RoboDK station: NiryoStation.rdk

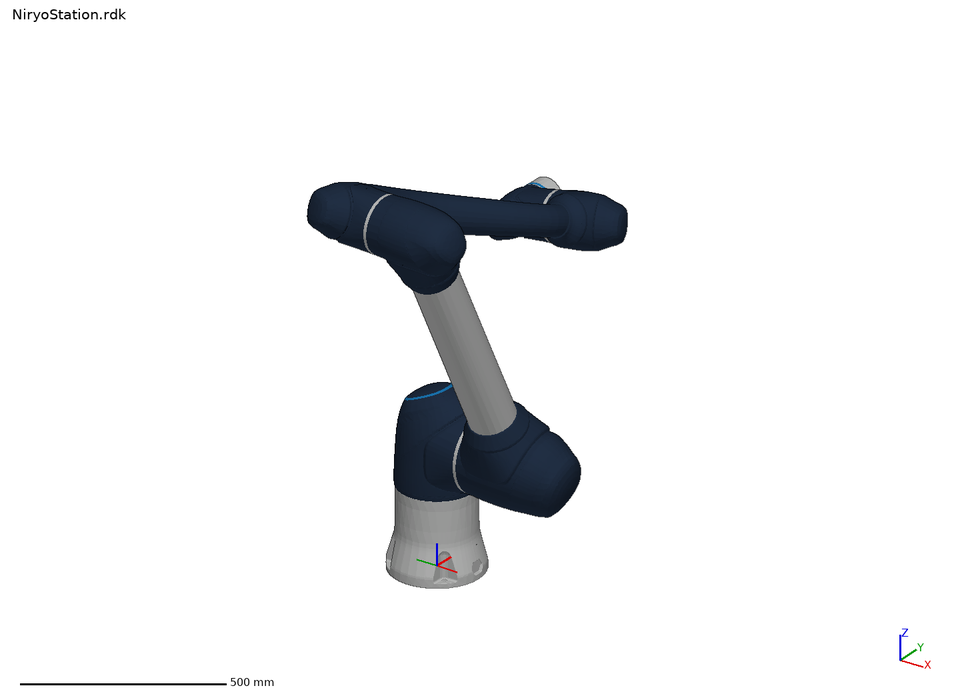
[picture v0: the station drawn from its stored meshes, robots at their saved joint values, targets as dots, program paths as lines]
Station NiryoStation (saved by RoboDK 5.5.1). Poses are relative to the parent item; angles as X-Y-Z fixed-axis rotations.
  - frame wall at (0, 0, 0) mm
    - frame RoboBase at (0, 0, 0) mm, rotated rx 0 ry 0 rz 90 deg
      - robot Doosan Robotics H2017: 6 axes, payload 20 kg, reach 1700 mm, repeatability 0.1 mm
          modified DH rows (alpha deg, a mm, theta deg, d mm): 0, 0, 180, 344.3; -90, 0, -90, -9.9; 0, 845, -90, 0; -90, 0, 0, 734; 90, 0, 0, 0; -90, 0, 180, 121
          joint limits [-360, -130, -160, -360, -360, -360] to [360, 130, 160, 360, 360, 360]; home [0, 0, -90, 0, 0, 0]; saved at [-183.549, 26.062, -136.98, -8.888, 22.786, -44.881]
  - Python program main (listed below)

--- Python program main ---
# Type help("robodk.robolink") or help("robodk.robomath") for more information
# Press F5 to run the script
# Documentation: https://robodk.com/doc/en/RoboDK-API.html
# Reference:     https://robodk.com/doc/en/PythonAPI/robodk.html
# Note: It is not required to keep a copy of this file, your Python script is saved with your RDK project


#Importing custom library
from setup import setup
from robot_comands import *
from import_plan import import_plan
from geometry import *


# Forward and backwards compatible use of the RoboDK API:
# Remove these 2 lines to follow python programming guidelines

#Important Observation: to the code to work, the reference frame of the robot must be the wall not the RobotBase

if __name__ == '__main__':

    print('Initiating robot position:')
    [RDK, robot] = ini_robot()#Iniciating Robot and RoboDK comunication
    [w,h,points_lists] = import_plan('C:\\Users\Fernando\Documents\Challenge\Imagine_Make\essaiim.csv')#Importing Plan


    print('Initiating Calibration Routine, please follow the intructions:')
    #RobotHeadFrame = setup(w,h,robot)#Calibration Function
    RobotHeadFrame = RefFrame(-420, -2570,840)

    print('End of calibration')
    print(f"Position to Robot's head in relation to the wall lower left corner: {RobotHeadFrame}\n")
    set_robot_frame(RDK,robot,RobotHeadFrame)#Updating Robot Frame

    print(f'Starting service...{len(points_lists)} operations to do')
    counter = 1

    for point in points_lists:#Pointing to all points
        print(f'Targenting {counter}° point {point} in wall')
        point_2_wall(RDK,robot, point)
        print('Press Enter to go to the next point\n')
        input()
        counter += 1

    print('Work done!! Congratulations =)')
